// TIA Portal project "Recipe_Manager" (V18)

(* hardware
DEVICE "S7-1500/ET200MP station_1"  S7-1500 station
   slot 0: "Rail_0"  Rack  6ES7 590-1***0-0AA0
DEVICE "S7-1500/ET200MP station_2"  S7-1500 station
   slot 0: "Rail_0"  Rack  6ES7 590-1***0-0AA0
   slot 1: "PLC_1"  CPU 1511-1 PN  6ES7 511-1AK02-0AB0  V2.8
      slot 3: "CPU display_1"  6ES7591-1AA00-0AA0
      slot 32768: "PROFINET interface_1"  X1
         slot 32769: "Port_1"  X1 P1
         slot 32770: "Port_2"  X1 P2
      slot 34817: "Virtual CP interface port_1"  Virtual CP interface port  Virtual CP interface port
   slot 2: "DI 16x24VDC BA_1"  DI 16x24VDC BA  6ES7 521-1BH10-0AA0  V1.1
   slot 3: "DQ 16x24VDC/0.5A BA_1"  DQ 16x24VDC/0.5A BA  6ES7 522-1BH10-0AA0  V1.1
*)

// ===== PLC "PLC_1"  CPU 1511-1 PN =====

VAR_GLOBAL   // PLC tag table "Default tag table"
   "Emitter_Enable" AT %Q0.0 : Bool;
   "Capper_Extend" AT %Q0.1 : Bool;
   "Labeler_Extend" AT %Q0.2 : Bool;
   "Remover_Enable" AT %Q0.3 : Bool;
   "Conveyor_Speed" AT %QD100 : Real;
   "Box_AtFill" AT %I0.0 : Bool;
   "Capper_FullExtend" AT %I0.1 : Bool;
   "Capper_FullRetract" AT %I0.2 : Bool;
   "Box_AtLabel" AT %I0.3 : Bool;
   "Labeler_FullExtend" AT %I0.4 : Bool;
   "Labeler_FullRetract" AT %I0.5 : Bool;
   "Tag_1" AT %MW102 : Word;
END_VAR

TYPE "Recipe_Type"
   STRUCT
      Product_Name : String := 'Product_A';
      Conveyor_Speed_Pct : Int := 50;
      Cap_Hold_Time : Int := 500;
      Label_Hold_Time : Int := 300;
      Batch_Count_Target : Int := 10;
      Recipe_Active : Bool;
   END_STRUCT;
END_TYPE

DATA_BLOCK "Recipe_DB"   // DB1
{ S7_Optimized_Access := 'FALSE' }
VERSION : 0.1
   VAR
      Recipes : Array[0..9] of "Recipe_Type";
   END_VAR
BEGIN
   Recipes[0].Product_Name := 'Water_500ml';
   Recipes[0].Conveyor_Speed_Pct := 60;
   Recipes[1].Product_Name := 'Juice_330ml';
   Recipes[1].Conveyor_Speed_Pct := 45;
   Recipes[1].Cap_Hold_Time := 400;
   Recipes[1].Label_Hold_Time := 250;
   Recipes[1].Batch_Count_Target := 15;
   Recipes[2].Product_Name := 'Oil_1L';
   Recipes[2].Conveyor_Speed_Pct := 25;
   Recipes[2].Cap_Hold_Time := 700;
   Recipes[2].Label_Hold_Time := 400;
   Recipes[2].Batch_Count_Target := 5;
END_DATA_BLOCK

DATA_BLOCK "Control_DB"   // DB2
{ S7_Optimized_Access := 'FALSE' }
VERSION : 0.1
   VAR
      Active_Recipe_Index : Int;
      Conveyor_Speed_Pct : Int := 50;
      Drive_Enable : Bool := true;
      Drive_Fault_Reset : Bool;
      Actual_Speed_Pct : Int;
      Product_Count : Int;
      Line_Running : Bool := true;
      Fault_Active : Bool;
      Active_Cap_Time : Int;
      Active_Label_Time : Int;
      Active_Batch_Target : Int;
   END_VAR
BEGIN
END_DATA_BLOCK

DATA_BLOCK "Modbus_Connection"   // DB3
{ S7_Optimized_Access := 'TRUE' }
VERSION : 0.1
   VAR
      Conn_Data : TCON_IP_v4;
   END_VAR
BEGIN
   Conn_Data.InterfaceId := 64;
   Conn_Data.ID := 1;
   Conn_Data.ConnectionType := 11;
   Conn_Data.LocalPort := 502;
END_DATA_BLOCK

DATA_BLOCK "Recipe_Control_DB_1"   // DB4
{ S7_Optimized_Access := 'FALSE' }
VERSION : 0.1
// stored: InstanceOfName Recipe_Control
"Recipe_Control"
BEGIN
END_DATA_BLOCK

FUNCTION_BLOCK "Recipe_Control"   // FB1, SCL
{ S7_Optimized_Access := 'FALSE' }
VERSION : 0.1
   VAR
      Cap_State : Int;
      Label_State : Int;
      Last_Recipe_Index : Int := -1;
      Label_Timer : TON_TIME;
      Cap_Timer : TON_TIME;
   END_VAR
BEGIN
   // =========================================================
   // Recipe_Control FB — FINAL MASTER CODE
   // =========================================================

   // ── 1. Auto-Load Recipe Timers from Database ──────────────
   "Control_DB".Active_Cap_Time := "Recipe_DB".Recipes["Control_DB".Active_Recipe_Index].Cap_Hold_Time;
   "Control_DB".Active_Label_Time := "Recipe_DB".Recipes["Control_DB".Active_Recipe_Index].Label_Hold_Time;

   // ── 2. ONE-SHOT: Auto-Load Speed ONLY on Recipe Change ────
   IF "Control_DB".Active_Recipe_Index <> #Last_Recipe_Index THEN
       // Grab the new speed from the database just this once
       "Control_DB".Conveyor_Speed_Pct := "Recipe_DB".Recipes["Control_DB".Active_Recipe_Index].Conveyor_Speed_Pct;

       // Update the memory so this block shuts off and lets the SCADA slider work
       #Last_Recipe_Index := "Control_DB".Active_Recipe_Index;
   END_IF;

   // ── 3. Stop everything when line is off ───────────────────
   IF NOT "Control_DB".Line_Running THEN
       "Capper_Extend" := FALSE;
       "Labeler_Extend" := FALSE;
       "Conveyor_Speed" := REAL#0.0;
       #Cap_State := 0;
       #Label_State := 0;
       #Cap_Timer(IN := FALSE,
                  PT := T#1ms);
       #Label_Timer(IN := FALSE,
                    PT := T#1ms);
       RETURN;
   END_IF;

   // ── 4. Emitter and Remover ────────────────────────────────
   "Emitter_Enable" := "Control_DB".Line_Running;
   "Remover_Enable" := "Control_DB".Line_Running;

   // ── 5. Cap pusher state machine (Sensor-Centering) ────────
   CASE #Cap_State OF

       0: // Waiting — belt running at SCADA slider speed
           "Capper_Extend" := FALSE;
           "Conveyor_Speed" := REAL#3.0 * INT_TO_REAL("Control_DB".Conveyor_Speed_Pct) / REAL#100.0;
           #Cap_Timer(IN := FALSE,
                      PT := T#1ms);

           // As soon as the sensor hits, instantly jump to Capping
           IF "Box_AtFill" THEN
               #Cap_State := 2;
           END_IF;

       2: // Stop belt and extend pusher — SCADA RECIPE HOLD TIME
           "Conveyor_Speed" := REAL#0.0;
           "Capper_Extend" := TRUE;
           #Cap_Timer(IN := TRUE,
                      PT := DINT_TO_TIME(INT_TO_DINT("Control_DB".Active_Cap_Time)));

           IF #Cap_Timer.Q THEN
               #Cap_Timer(IN := FALSE,
                          PT := T#1ms);
               #Cap_State := 3;
           END_IF;

       3: // Retract pusher
           "Conveyor_Speed" := REAL#0.0;
           "Capper_Extend" := FALSE;
           #Cap_Timer(IN := TRUE,
                      PT := T#800ms);
           IF #Cap_Timer.Q THEN
               #Cap_Timer(IN := FALSE,
                          PT := T#1ms);
               #Cap_State := 4;
           END_IF;

       4: // Wait for box to clear then resume at SCADA slider speed
           "Conveyor_Speed" := REAL#3.0 * INT_TO_REAL("Control_DB".Conveyor_Speed_Pct) / REAL#100.0;
           "Capper_Extend" := FALSE;
           #Cap_Timer(IN := TRUE,
                      PT := T#1500ms);
           IF #Cap_Timer.Q AND NOT "Box_AtFill" THEN
               #Cap_Timer(IN := FALSE,
                          PT := T#1ms);
               #Cap_State := 0;
           END_IF;

   END_CASE;

   // ── 6. Label pusher state machine (Sensor-Centering) ──────
   CASE #Label_State OF

       0: // Waiting — belt running
           "Labeler_Extend" := FALSE;
           #Label_Timer(IN := FALSE,
                        PT := T#1ms);

           // As soon as the sensor hits, instantly jump to Labeling
           IF "Box_AtLabel" THEN
               #Label_State := 2;
           END_IF;

       2: // Extend pusher and hold — SCADA RECIPE HOLD TIME
           "Labeler_Extend" := TRUE;
           #Label_Timer(IN := TRUE,
                        PT := DINT_TO_TIME(INT_TO_DINT("Control_DB".Active_Label_Time)));

           IF #Label_Timer.Q THEN
               #Label_Timer(IN := FALSE,
                            PT := T#1ms);
               "Control_DB".Product_Count := "Control_DB".Product_Count + 1;
               #Label_State := 3;
           END_IF;

       3: // Retract pusher
           "Labeler_Extend" := FALSE;
           #Label_Timer(IN := TRUE,
                        PT := T#800ms);
           IF #Label_Timer.Q THEN
               #Label_Timer(IN := FALSE,
                            PT := T#1ms);
               #Label_State := 4;
           END_IF;

       4: // Wait for box to clear then reset
           "Labeler_Extend" := FALSE;
           #Label_Timer(IN := TRUE,
                        PT := T#1500ms);
           IF #Label_Timer.Q AND NOT "Box_AtLabel" THEN
               #Label_Timer(IN := FALSE,
                            PT := T#1ms);
               #Label_State := 0;
           END_IF;

   END_CASE;
END_FUNCTION_BLOCK

ORGANIZATION_BLOCK "Main"   // OB1, LAD, ProgramCycle
TITLE = "Main Program Sweep (Cycle)"
{ S7_Optimized_Access := 'TRUE' }
VERSION : 0.1
   VAR_INPUT
      Initial_Call : Bool;   // Initial call of this OB
      Remanence : Bool;   // =True, if remanent data are available
   END_VAR
BEGIN

REGION Network 1
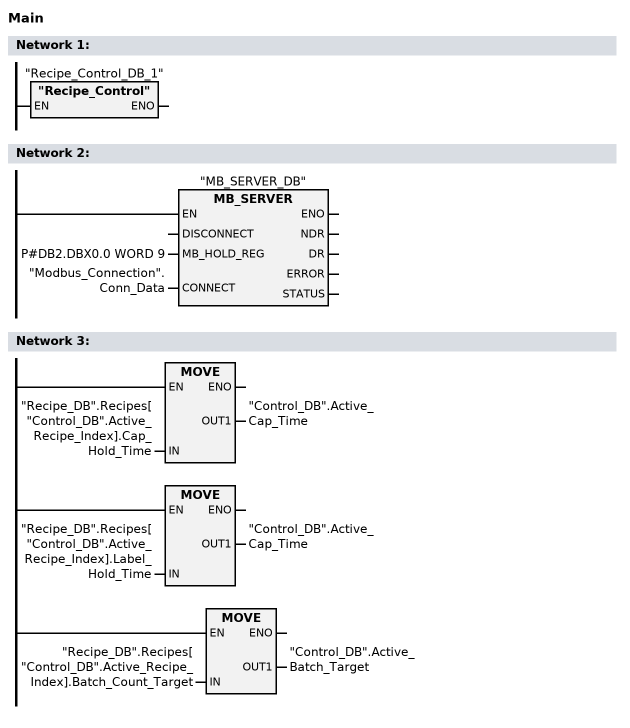
   RUNG wire#powerrail
      "Recipe_Control_DB_1"()
   END_RUNG
   // the same network as SCL:
   "Recipe_Control_DB_1"();   // "Recipe_Control"
END_REGION

REGION Network 2
   "MB_SERVER_DB"(MB_HOLD_REG := P#DB2.DBX0.0 WORD 9, CONNECT := "Modbus_Connection".Conn_Data);   // MB_SERVER
END_REGION

REGION Network 3
   RUNG wire#powerrail
      Move(in := "Recipe_DB".Recipes["Control_DB".Active_Recipe_Index].Cap_Hold_Time, out1 => "Control_DB".Active_Cap_Time)
   END_RUNG
   RUNG wire#powerrail
      Move(in := "Recipe_DB".Recipes["Control_DB".Active_Recipe_Index].Label_Hold_Time, out1 => "Control_DB".Active_Cap_Time)
   END_RUNG
   RUNG wire#powerrail
      Move(in := "Recipe_DB".Recipes["Control_DB".Active_Recipe_Index].Batch_Count_Target, out1 => "Control_DB".Active_Batch_Target)
   END_RUNG
   // the same network as SCL:
   "Control_DB".Active_Cap_Time := "Recipe_DB".Recipes["Control_DB".Active_Recipe_Index].Cap_Hold_Time;
   "Control_DB".Active_Cap_Time := "Recipe_DB".Recipes["Control_DB".Active_Recipe_Index].Label_Hold_Time;
   "Control_DB".Active_Batch_Target := "Recipe_DB".Recipes["Control_DB".Active_Recipe_Index].Batch_Count_Target;
END_REGION
END_ORGANIZATION_BLOCK